// LS Electric XG5000 project: 동남98
// PLC NewPLC
// module base 0 slot 0: 입출력 모듈:XBC-DN/DP14E (DC 24V 입력 8점, 트랜지스터 출력 6점)

PROGRAM NewProgram (task: 스캔 프로그램)

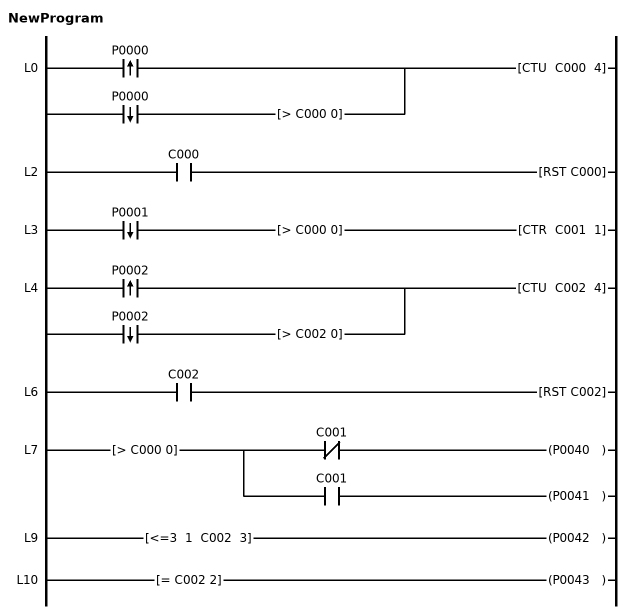
; L0
LOADP     P0000
LOADN     P0000
AND>      C000 0
OR LOAD
CTU       C000 4
; L2
LOAD      C000
RST       C000
; L3
LOADN     P0001
AND>      C000 0
CTR       C001 1
; L4
LOADP     P0002
LOADN     P0002
AND>      C002 0
OR LOAD
CTU       C002 4
; L6
LOAD      C002
RST       C002
; L7
LOAD>     C000 0
MPUSH
AND NOT   C001
OUT       P0040
MPOP
AND       C001
OUT       P0041
; L9
LOAD<=3   1 C002 3
OUT       P0042
; L10
LOAD=     C002 2
OUT       P0043